PROGRAM TCPTimeOut
VAR
	fbLocalTime : FB_LocalSystemTime;
	iPreviousTime : WORD := 0;
END_VAR


fbLocalTime(
	sNetId := ,
	bEnable := TRUE,
	dwCycle := 10,
	dwOpt := ,
	tTimeout := DEFAULT_ADS_TIMEOUT,
);

	IF fbLocalTime.systemTime.wMilliseconds - iPreviousTime >= 200 THEN	
		GVL_SAFETY.SafetyTriggerd := TRUE;	
	END_IF
	
	IF RunTCP.sCommand > '' THEN
		iPreviousTime := fbLocalTime.systemTime.wMilliseconds;
	END_IF

END_PROGRAM

(* stored: Version 1.1.0.1, ProductVersion 3.1.4024.3
   POU TCPTimeOut: Id {e0e15d90-c382-4ea1-a8cf-110410e3e3f5}, SpecialFunc None *)
